// TIA Portal V20 export
FUNCTION_BLOCK "CentralShifter_AutoDrive"   // FB11, LAD
{ S7_Optimized_Access := 'TRUE' }
// stored: MemoryReserve 100, SetENOAutomatically false
   VAR_INPUT
      Destination_Pos : DInt;
      Actual_Pos : DInt;
      Drive_To_Pos : Bool;
   END_VAR
   VAR_OUTPUT
      Auto_Speed : Real;
      Auto_Drive_Forward : Bool;
      Auto_Drive_Backward : Bool;
      Deceleration : Real;
   END_VAR
   VAR
      distance : DInt;
      tolerance : Real := 4.0;
      prevSpeed : Real;
      StartSpeed : Real := 380.0;
      EndSpeed : Real := 75.0;
      DecelTimer : TON_TIME;
      progress { S7_SetPoint := 'True'} : Real;
      StopRampTimer : TON_TIME;
      RampActive { S7_SetPoint := 'True'} : Bool;
      LastDirection : Int;
      StopProgress : Real;
      Vel_To_Stop : Real;
      Drive_To_Pos_Last : Bool;
      StopRampTimer_1 : TON_TIME;
      DriveOffTimer { S7_SetPoint := 'True'} : TON_TIME;
   END_VAR
BEGIN

REGION Network 1 (SCL)
   #distance := ABS(#Destination_Pos - #Actual_Pos);

   // --- wykrywanie zbocza opadającego przycisku ---
   IF NOT #Drive_To_Pos AND #Drive_To_Pos_Last THEN
       // Po puszczeniu przycisku — aktywuj rampę (jeśli jest poza tolerancją)
       IF #distance > #tolerance THEN
           #RampActive := TRUE;
           #StopRampTimer(IN := TRUE,
                          PT := T#2s); // 2 sekundy rampy
           #Vel_To_Stop := "CS_Drive_PL".Velocity; // zapamiętaj prędkość do wyhamowania
       ELSE
           // Jeśli już w tolerancji — od razu stop
           #RampActive := FALSE;
           #StopRampTimer.IN :=0;
           #Auto_Speed := 0.0;
           #Auto_Drive_Forward := FALSE;
           #Auto_Drive_Backward := FALSE;
       END_IF;
   END_IF;

   #Drive_To_Pos_Last := #Drive_To_Pos;

   // --- Główna logika ruchu ---
   IF #Drive_To_Pos THEN
       // --- Tryb aktywnego ruchu ---
       IF #distance <= #tolerance THEN
           "HMI_Central_Shifter".CS_Status_Auto_Go_to_Des := 2;
           #Auto_Drive_Forward := FALSE;
           #Auto_Drive_Backward := FALSE;
           #Auto_Speed := 0.0;
           #DecelTimer.IN := FALSE;
       ELSE
           "HMI_Central_Shifter".CS_Status_Auto_Go_to_Des := 1;

           // Kierunek
           IF #Actual_Pos > #Destination_Pos THEN
               #Auto_Drive_Forward := TRUE;
               #Auto_Drive_Backward := FALSE;
               #LastDirection := 1;
           ELSE
               #Auto_Drive_Forward := FALSE;
               #Auto_Drive_Backward := TRUE;
               #LastDirection := -1;
           END_IF;

           // Rampowanie w zależności od odległości
           IF #distance > 5000.0 THEN
               #Auto_Speed := #StartSpeed;
               #DecelTimer.IN := FALSE;
           ELSE
               #DecelTimer(IN := TRUE,
                           PT := T#5s);
               #progress := (5000.0 - #distance) / 5000.0;
               IF #progress > 1.0 THEN
                   #progress := 1.0;
               END_IF;
               #Auto_Speed := #StartSpeed - #progress * (#StartSpeed - #EndSpeed);
           END_IF;
       END_IF;

       // Reset rampy podczas aktywnego ruchu
       #RampActive := FALSE;
       #StopRampTimer.IN := FALSE;

   ELSE
       // --- Tryb hamowania rampą po puszczeniu przycisku ---
       IF #RampActive THEN
           #StopProgress := INT_TO_REAL(TIME_TO_INT(#StopRampTimer.ET)) / INT_TO_REAL(TIME_TO_INT(T#2s));
           IF #StopProgress > 1.0 THEN
               #StopProgress := 1.0;
           END_IF;

           // Liniowe zmniejszanie prędkości
           #Auto_Speed := (1.0 - #StopProgress) * #Vel_To_Stop;

           // Kierunek zgodny z ostatnim
           IF #LastDirection = 1 THEN
               #Auto_Drive_Forward := TRUE;
               #Auto_Drive_Backward := FALSE;
           ELSIF #LastDirection = -1 THEN
               #Auto_Drive_Forward := FALSE;
               #Auto_Drive_Backward := TRUE;
           ELSE
               #Auto_Drive_Forward := FALSE;
               #Auto_Drive_Backward := FALSE;
           END_IF;

           // Po zakończeniu rampy
           IF #StopRampTimer.Q THEN
               #Auto_Speed := 0.0;
               #Auto_Drive_Forward := FALSE;
               #Auto_Drive_Backward := FALSE;
               #RampActive := FALSE;
               #StopRampTimer.IN :=0;
               #LastDirection := 0;
           END_IF;
       ELSE
           // Jeśli rampa nieaktywna — wymuszone zatrzymanie
           #Auto_Speed := 0.0;
           #Auto_Drive_Forward := FALSE;
           #Auto_Drive_Backward := FALSE;
           #StopRampTimer.IN := FALSE;
       END_IF;
   END_IF;

   // --- Status ---
   IF #distance <= #tolerance THEN
       "HMI_Central_Shifter".CS_Status_Auto_Go_to_Des := 2;
   ELSIF #Drive_To_Pos THEN
       "HMI_Central_Shifter".CS_Status_Auto_Go_to_Des := 1;
   ELSE
       "HMI_Central_Shifter".CS_Status_Auto_Go_to_Des := 0;
   END_IF;



   // --- Granice bezpieczeństwa ---
   IF #Actual_Pos <= 0 THEN
       #Auto_Drive_Forward := FALSE;
       #Auto_Drive_Backward := FALSE;
       #Auto_Speed := 0.0;
       #DecelTimer.IN := FALSE;
       #RampActive := FALSE;
       #StopRampTimer.IN := FALSE;
   END_IF;
END_REGION
END_FUNCTION_BLOCK
